// TIA Portal V20 export
TYPE "LER_typeUnitResultData"
// stored: Access Published
   STRUCT
      hotPressLeft { ExternalWritable := 'False'} : "LER_typeServoPressTrackingData";
      hotPressRight { ExternalWritable := 'False'} : "LER_typeServoPressTrackingData";
      hipotThicknesPress { ExternalWritable := 'False'} : "LER_typeServoPressTrackingData";
      hipot { ExternalWritable := 'False'} : "LER_typeHipotTrackingData";
      thickness { ExternalWritable := 'False'} : "LER_typeThicknessTrackingData";
      vision { ExternalWritable := 'False'} : "LER_typeVisionTrackingData";
      laserMarker { ExternalWritable := 'False'} : "LER_typeLaserMarkTrackingData";
      qrFixReader { ExternalWritable := 'False'} : "LER_typeQrReadTrackingData";
      weightChecker { ExternalWritable := 'False'} : "LER_typeWeightCheckTrackingData";
   END_STRUCT;
END_TYPE
